FUNCTION_BLOCK Safety
VAR_INPUT	
END_VAR
VAR_OUTPUT
END_VAR
VAR
	{attribute 'OPC.UA.DA' := '0'}
	_message : StringBuilder;
	{attribute 'OPC.UA.DA' := '0'}
	_logger : Logger;
	
	{attribute 'OPC.UA.DA' := '0'}
	_execStartSafety : BOOL := TRUE;	
	{attribute 'OPC.UA.DA' := '0'}
	_execErrAcq : BOOL; 

	{attribute 'OPC.UA.DA' := '0'}
	GroupComErr AT %I* : BOOL;
	{attribute 'OPC.UA.DA' := '0'}
	GroupComStartup AT %I* : BOOL;
	{attribute 'OPC.UA.DA' := '0'}
	GroupFBDeactivate AT %I* : BOOL;
	{attribute 'OPC.UA.DA' := '0'}
	GroupFBErr AT %I* : BOOL;
	{attribute 'OPC.UA.DA' := '0'}
	GroupFBRun AT %I* : BOOL;
	{attribute 'OPC.UA.DA' := '0'}
	GroupInRun AT %I* : BOOL;
	{attribute 'OPC.UA.DA' := '0'}
	GroupOtherErr AT %I* : BOOL;
	{attribute 'OPC.UA.DA' := '0'}
	GroupOutErr AT %I* : BOOL;	 
	{attribute 'OPC.UA.DA' := '0'}
	GroupModuleFault AT %Q* : BOOL;
	{attribute 'OPC.UA.DA' := '0'}
	GroupStartStop AT %Q* : BOOL;
	{attribute 'OPC.UA.DA' := '0'}	
	GroupErrAck AT %Q* : BOOL;

	{attribute 'OPC.UA.DA' := '0'}
	_pulseGenerator : TON;	
	{attribute 'OPC.UA.DA' := '0'}
	_itemScheduler : INT;
	
END_VAR


IF NOT GroupInRun THEN
	IF _pulseGenerator.Q THEN
		_pulseGenerator(IN := FALSE, PT := T#10MS);
			
		CASE _itemScheduler OF					
			0:	IF NOT GroupFBRun THEN
					_logger.Information(_message.Reset().Append('Safety: started').ToString());
					GroupStartStop := TRUE;	
				END_IF
				_itemScheduler := 1;
	
			1:	IF NOT GroupErrAck THEN
					GroupErrAck := TRUE;
				END_IF
				_itemScheduler := 2;
	
			2:  IF GroupErrAck THEN
					GroupErrAck := FALSE;
					_logger.Information(_message.Reset().Append('Error acknowledgement: executed').ToString());
				END_IF
				_itemScheduler := 0;
		END_CASE
	ELSE
		_pulseGenerator(IN := TRUE, PT := T#1000MS);		
	END_IF
END_IF

END_FUNCTION_BLOCK

(* stored: Version 1.1.0.1, ProductVersion 3.1.4024.12
   POU Safety: Id {747e9edb-099e-48be-8648-a964116c48d6}, SpecialFunc None *)
